TYPE STATE:
    STRUCT
        curTime: REAL;
    END_STRUCT;
END_TYPE
